PROGRAM CraneSimulation
VAR
	fTime : LREAL; 	
	bRunning : BOOL;
	fPositionAutoMode : LREAL; 
	fInitialPosition : LREAL; 
	fInitialVelocity : LREAL; 
	eStatus : E_Status; 
	eMode : E_Mode; 
	paramCylinderPiston : REFERENCE TO ST_pCylinderPiston;
	fMaxPistonStroke : LREAL;
END_VAR

IF Inputs.bStartSimulation AND Inputs.bAutoMode  THEN
	fTime := fTime + Parameters.fCyclicTime;
ELSE
	fTime := 0; 	
END_IF

IF fTime > 0 AND Inputs.bAutoMode THEN 
	bRunning := TRUE;
ELSE
	bRunning := FALSE;
END_IF

fPositionAutoMode := Inputs.fCylinderVelocityReference * 1/2*(fTime*fTime) + fInitialVelocity * fTime + fInitialPosition;

// added max/min outout value to avoid to large output for visualization
IF fPositionAutoMode >= Parameters.pCylinderPiston.fPistonPosMax THEN
	fPositionAutoMode := Parameters.pCylinderPiston.fPistonPosMax;	
ELSIF fPositionAutoMode <= Parameters.pCylinderPiston.fPistonPosMin  THEN
	fPositionAutoMode := Parameters.pCylinderPiston.fPistonPosMin; 
ELSE	
	fPositionAutoMode := fPositionAutoMode;
END_IF

IF Inputs.bAutoMode THEN
	Outputs.fCylinderPosition := fPositionAutoMode;
ELSE
	Outputs.fCylinderPosition := Inputs.fManualCylinderPositionReference;	
END_IF

Outputs.bSimulationRunning := bRunning;  
Outputs.fSimulationTime := fTime; 
Outputs.fCylinderVelocity := Inputs.fCylinderVelocityReference;
Outputs.pt1_y := LREAL_TO_INT(Outputs.fCylinderPosition * Parameters.pCylinderPiston.fPistonScale);



// Status

IF Inputs.bEnableSimulation THEN
	eStatus := E_Status.Ready;
ELSE 
	eStatus := E_Status.Fault;	
END_IF

IF Inputs.bStartSimulation THEN
	eStatus := E_Status.Starting;
END_IF

IF bRunning THEN
	eStatus := E_Status.Running;
END_IF

// Mode
IF Inputs.bAutoMode THEN
	eMode := E_Mode.Auto;
ELSE 
	eMode := E_Mode.Manual;	
END_IF

paramCylinderPiston.fPistonPosMax := fMaxPistonStroke;

END_PROGRAM

(* stored: Version 1.1.0.1, ProductVersion 3.1.4024.10
   POU CraneSimulation: Id {c255987f-7a58-4573-9ac9-545c12e8d4a5}, SpecialFunc None *)
